{attribute 'qualified_only'}
{attribute 'strict'}
TYPE DatabaseStep :
(
	RESET,
	DISCONNECT, 
	CONNECT, 
	IDLE, 
	EXECUTE, 
	LOAD_DATA,
	
	size
);
END_TYPE

(* stored: Version 1.1.0.1, ProductVersion 3.1.4024.11
   DUT DatabaseStep: Id {4f0478fb-5e04-4f47-9d68-c17e362bb47d} *)
